FUNCTION FKT_Scale : LREAL
VAR_INPUT
	// Unterer Auflösungsbereich
	X1: LREAL;
	// Oberer Auflösungsbereich
	X2: LREAL;
	// Unterer Darstellungsbereich
	Y1: LREAL;
	// Oberer Darstellungsbereich
	Y2: LREAL;
END_VAR
VAR
	// Rohwert in Real
	X: LREAL;
	// Skalierter Messwert
	Y: LREAL := 0;
END_VAR
VAR_INPUT
	// Analoger Eingang in 12 bzw. 16 Bit
	Rohwert: LREAL;
END_VAR

X := Rohwert;

Y := ((((Y2-Y1)/(X2-X1))*(X-X1))+Y1);			// Skalierung über eine lineare Funktion

IF Y > Y2 THEN
	Y := Y2;									// Obere Begrenzung
ELSIF Y < Y1 THEN
	Y := Y1;									// Untere Begrenzung
END_IF

FKT_Scale := Y;									// Ausgabe

END_FUNCTION

(* stored: Version 1.1.0.1, ProductVersion 3.1.4024.6
   POU FKT_Scale: Id {f23a5b1a-922f-4610-8905-a8549e0de617}, SpecialFunc None *)
